INTERFACE I_ListOfTests

METHOD AddTest
VAR_INPUT
    Test : I_UnitTest;
END_VAR
END_METHOD

PROPERTY Count : DINT
GET
END_GET
END_PROPERTY

METHOD FindTestIndex : DINT
VAR_INPUT
	Test : I_UnitTest;
END_VAR
END_METHOD

METHOD GetTest : I_UnitTest
VAR_INPUT
    Index : DINT;
END_VAR
END_METHOD

METHOD SetTest : I_UnitTest
VAR_INPUT
    Test : I_UnitTest;
    Index : DINT;
END_VAR
END_METHOD

PROPERTY TestGroupName : T_MaxString
GET
END_GET
END_PROPERTY

END_INTERFACE

(* stored: Version 1.1.0.1, ProductVersion 3.1.4024.11
   Itf I_ListOfTests: Id {893e7e43-a7a7-456e-9517-e3d21b74d5fa}
   Method AddTest: Id {e9ad3765-0af3-47ea-a604-b236c0477164}
   Property Count: Id {cd9ef367-f066-49ff-883b-2dba33c01866}
   Get Get: Id {b7f24ab7-3fd8-4494-9397-81af06512e9e}
   Method FindTestIndex: Id {ef55a53b-f2a4-443d-a008-5ccaec33d191}
   Method GetTest: Id {bc5e0acc-0aa8-4117-b203-55864887c248}
   Method SetTest: Id {f50ad0a9-50fa-4169-af3d-919c413751b1}
   Property TestGroupName: Id {64854b96-8b20-4b92-aaa4-265f6f43b2cd}
   Get Get: Id {36f61fd4-09fe-4755-a67d-d4ee53f9e0c3} *)
